Omron CX-Programmer project 新規ﾌﾟﾛｼﾞｪｸﾄ (CX-Programmer 9.61)

# PLC hoge1: CP1L L

## Program 新規ﾌﾟﾛｸﾞﾗﾑ1 (cyclic task 0)
Local symbols
I 0.00 BOOL
Q 100.00 BOOL

### Section ｾｸｼｮﾝ1

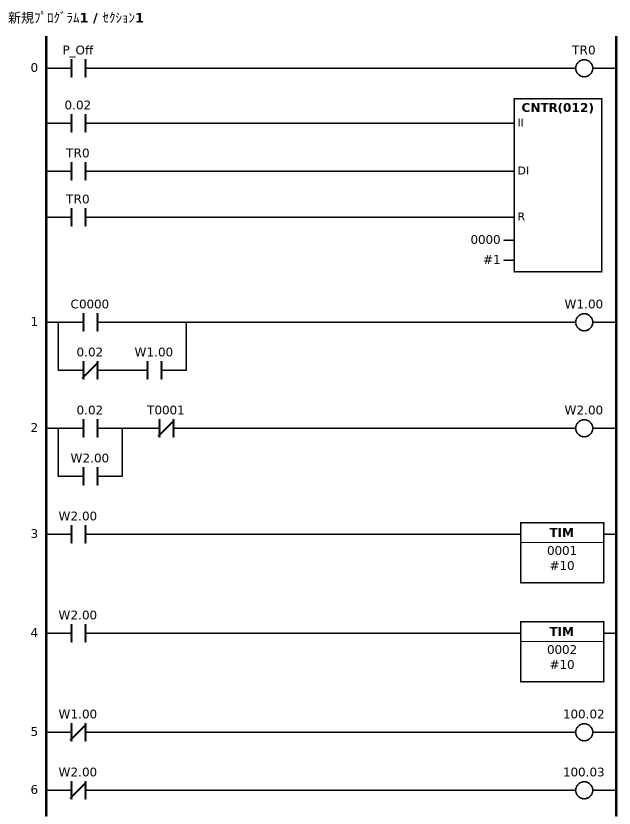
; rung 0
LD 0.02
LD P_Off
OUT TR0
LD TR0
CNTR(012) 0000 #1
; rung 1
LD C0000
LDNOT 0.02
AND W1.00
ORLD
OUT W1.00
; rung 2
LD 0.02
OR W2.00
ANDNOT T0001
OUT W2.00
; rung 3
LD W2.00
TIM 0001 #10
; rung 4
LD W2.00
TIM 0002 #10
; rung 5
LDNOT W1.00
OUT 100.02
; rung 6
LDNOT W2.00
OUT 100.03

### Section END
; rung 0
END(001)